Yaskawa INFORM job: PKT.JBI

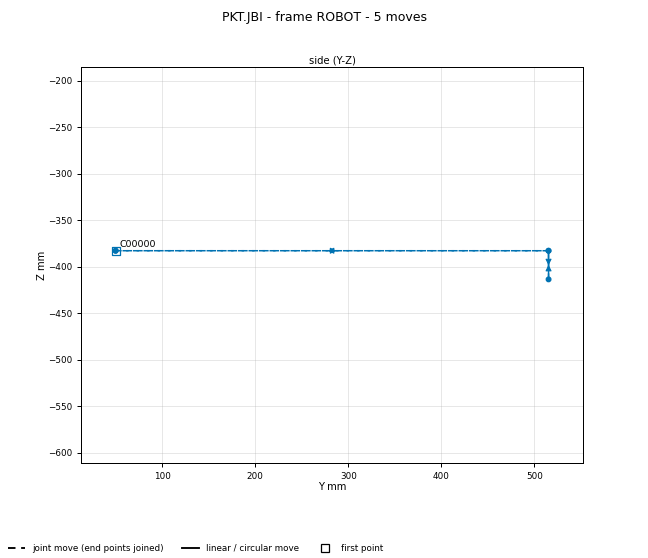
[picture p0: tool path of PKT.JBI in frame ROBOT, 5 of 5 moves have a stored position in this frame; points joined in program order, loops and branches not executed]
/JOB
//NAME PKT
//POS
///NPOS 5,5,0,0,0,0
///TOOL 0
///POSTYPE ROBOT
///RECTAN
///RCONF 1,0,1,0,0,0,0,0,0,0,0,0,0,0,0,0,0,0,0,0,0,0,0,0
C00000=1241.304,49.757,-382.806,0.2164,1.0287,-0.9640
C00001=1241.313,515.358,-382.818,0.2164,1.0280,-0.9641
C00002=1241.289,515.404,-413.622,0.2192,1.0285,-0.9656
C00003=1241.313,515.358,-382.818,0.2164,1.0280,-0.9641
C00004=1241.304,49.757,-382.806,0.2164,1.0287,-0.9640
///RCONF 0,0,0,0,0,0,0,0,0,0,0,0,0,0,0,0,0,0,0,0,0,0,0,0
BC00000=0.013
BC00001=0.013
BC00002=0.013
BC00003=0.013
BC00004=0.013
//INST
///DATE 2024/08/13 14:11
///ATTR SC,RW,RJ
////FRAME ROBOT
///GROUP1 RB1,BS1
NOP
MOVJ C00000 BC00000 VJ=5.00
MOVJ C00001 BC00001 VJ=5.00
MOVL C00002 BC00002 V=25.0  //1
MOVJ C00003 BC00003 VJ=5.00
MOVJ C00004 BC00004 VJ=5.00
END
